TYPE CM_Valve_ALM :
STRUCT
END_STRUCT
END_TYPE

(* stored: Version 1.1.0.1, ProductVersion 3.1.4024.12
   DUT CM_Valve_ALM: Id {b199d886-454a-4533-9869-2f1bb3da657a} *)
